FUNCTION_BLOCK PUBLIC FB_RollingAverageTime
VAR_INPUT
	fInputValue	: TIME ; // Input value [Anny_Number] 
END_VAR
VAR_IN_OUT
	bNewValue		: BOOL ; // Add value to array (set back to false)
	arTimeValues 	: ARRAY [*] OF TIME ; // Array of LREAL values, from thich to get the average
END_VAR
VAR_OUTPUT
	fAverage	: TIME ; // Everage of entries
END_VAR
VAR
	nWriteIndex			: DINT := 0;
	nArrayUpperBound 	: DINT;
	nArrayLowerBound 	: DINT;
	
	reNewValue	: R_TRIG ; // New value trigger
END_VAR

// determine array boundries
nArrayLowerBound := LOWER_BOUND(arTimeValues,1);
nArrayUpperBound := LOWER_BOUND(arTimeValues,1);

// Check if nwrite index is within array bounds
nWriteIndex := LIMIT(nArrayLowerBound, nWriteIndex, nArrayUpperBound);

// Add value to Array 
reNewValue(CLK := bNewValue);
IF reNewValue.Q THEN
	arTimeValues[nWriteIndex] := fInputValue;
	IF nWriteIndex = nArrayUpperBound THEN
		nWriteIndex := nArrayLowerBound;
	ELSE
		nWriteIndex := nWriteIndex +1;
	END_IF
END_IF 

// Calculate average value 
fAverage := F_AverageTime(arTimeValues);

METHOD PUBLIC Cmd_Reset : BOOL
VAR_INPUT
END_VAR
MEMSET(destAddr := ADR(arTimeValues), 0, n := SIZEOF(arTimeValues));
Cmd_Reset := true;
END_METHOD

END_FUNCTION_BLOCK

(* stored: Version 1.1.0.1, ProductVersion 3.1.4024.9
   POU FB_RollingAverageTime: Id {2ed85561-b45d-4c2d-a6c8-63ae1fcecab1}, SpecialFunc None
   Method Cmd_Reset: Id {70f5173e-7280-468b-88a9-2af528650c8e} *)
